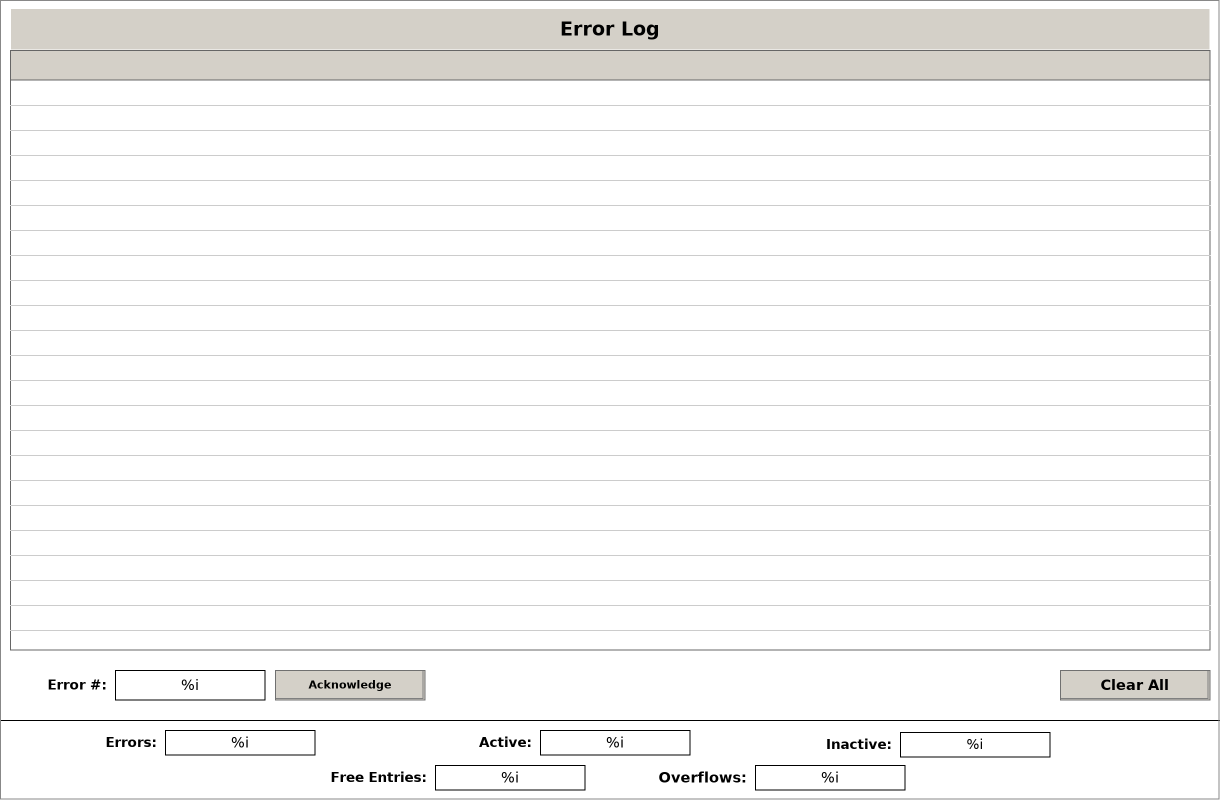
VISUALIZATION Error_Log_Visu  // 1220x800
    Table (10,50 1200x600), data array: MAIN.fbErrorSystem.ErrorSystem.aErrorData
        p1128707560: cSizeOfErrorData
        p1137915858: MAIN.fbErrorSystem.nTableRowIndex
        p1822360349: MAIN.fbErrorSystem.bValidSelection
        p3854506369: MAIN.fbErrorSystem.ErrorSystem.aErrorData[INDEX].ErrorNum
        p1892666644: MAIN.fbErrorSystem.ErrorSystem.aErrorData[INDEX].ErrorState
        p338671338: MAIN.fbErrorSystem.ErrorSystem.aErrorData[INDEX].iTerminalID
        p2170511999: MAIN.fbErrorSystem.ErrorSystem.aErrorData[INDEX].sDateTimeOn
        p3723444502: MAIN.fbErrorSystem.ErrorSystem.aErrorData[INDEX].sDateTimeOff
        p1218418051: MAIN.fbErrorSystem.ErrorSystem.aErrorData[INDEX].sErrorMessage
        p746581629: MAIN.fbErrorSystem.ErrorSystem.aErrorData[INDEX].ErrorPriority
        p2232123230: Error #
        p1755163831: Terminal ID
        p4092479075: Encountered on:
        p2237128397: Disapeared on:
        p505689113: Description
    Rectangle (11,9 1198x40), "Error Log"
    Button (275,670 150x30), "Acknowledge"
        tap MAIN.fbErrorSystem.bACK
        OnMouseUp: execute { MAIN.fbErrorSystem.nErrorNum := 0; }
    Button (1060,670 150x30), "Clear All"
        tap MAIN.fbErrorSystem.bReset
    Label (10,670 100x30), "Error #:"
    RoundedRectangle (115,670 150x30), "%i", text variable: MAIN.fbErrorSystem.nSelectedError
        OnMouseUp: write MAIN.fbErrorSystem.nErrorNum via Default, min 0
    Line (0,720) (1220,720)
    Label (10,730 150x25), "Errors:"
    Label (280,765 150x25), "Free Entries:"
    Label (600,765 150x25), "Overflows:"
    RoundedRectangle (165,730 150x25), "%i", text variable: MAIN.fbErrorSystem.ErrorSystem.nNoError
    RoundedRectangle (435,765 150x25), "%i", text variable: MAIN.fbErrorSystem.nFreePos
    RoundedRectangle (755,765 150x25), "%i", text variable: MAIN.fbErrorSystem.ErrorSystem.nNoOverflow
    Label (385,730 150x25), "Active:"
    Label (745,732 150x25), "Inactive:"
    RoundedRectangle (540,730 150x25), "%i", text variable: MAIN.fbErrorSystem.ErrorSystem.nNoActive
    RoundedRectangle (900,732 150x25), "%i", text variable: MAIN.fbErrorSystem.ErrorSystem.nNoInactive
END_VISUALIZATION

(* stored: Version 1.1.0.1, ProductVersion 3.1.4024.0
   Visu Error_Log_Visu: Id {58d8d61f-4113-4c1e-b3cb-a3d1b2e77b2d} *)
